PROGRAM MAIN
VAR
    // Clean slate - no variables needed here for now!
END_VAR

// Unconditionally call the background power and homing hardware engine
PRG_Hardware();
PRG_Manual_Drive();

END_PROGRAM

(* stored: Version 1.1.0.1, ProductVersion 3.1.4024.12
   POU MAIN: Id {c544dac8-e7b8-483c-93d1-a46857f04ac3}, SpecialFunc None *)
